// TIA Portal V19 export
TYPE "IF_TA1612_TTxNest"
   STRUCT
      OP : "OP_Int";
      Commands : "IF_Commands";
      "IF" : "IF_TA1612";
   END_STRUCT;
END_TYPE
